TYPE Mus_Sounds :
STRUCT
	note : E_Notes;
	tempo: INT;
END_STRUCT
END_TYPE

(* stored: Version 1.1.0.1, ProductVersion 3.1.4024.6
   DUT Mus_Sounds: Id {8a9d761e-c8b4-4123-81c0-568e5f53b9f7} *)
